// TIA Portal V21 export
DATA_BLOCK "Cabinets_Config"   // DB8
{ S7_Optimized_Access := 'TRUE' }
// stored: MemoryReserve 100
   VAR
      C0 : Array[1.."K_MaxCabinetNumber"] of "TypeC0";
   END_VAR
BEGIN
   C0[1].Power_L2_Disabled := false;
   C0[1].Power_L4_Disabled := false;
   C0[1].Safety_Z2_Disabled := true;
   C0[1].Safety_Z4_Disabled := false;
   C0[1].HWCombiNumber := 1;
   C0[2].HWCombiNumber := 3;
   C0[3..4].HWCombiNumber := 1;
END_DATA_BLOCK
